PROGRAM P1_01_Recipe
VAR
	i						:INT;
END_VAR

Recipes.Production.stPhase[1].bEnable := TRUE;
Recipes.Production_Phase_HMI.bEnable := TRUE;

Recipes.Production.iActivePhase := 0;

FOR i := 1 TO 20 DO
	IF Recipes.Production.stPhase[i].bEnable THEN
		Recipes.Production.iActivePhase := i;
	END_IF
	
	IF NOT Recipes.Production.stPhase[i].bEnable THEN
		Recipes.Production.stPhase[i] := Recipes.Production_Empty.stPhase[0];
	END_IF
END_FOR

END_PROGRAM

(* stored: Version 1.1.0.1
   POU P1_01_Recipe: Id {79a47d75-5839-4eec-98f3-898150a8f442}, SpecialFunc None *)
